// Mitsubishi GX Works2 project: 5   PLC: FX3U/FX3UC

// task Task_01 (event TRUE, interval 0, priority 31): POU_01

PROGRAM POU_01
VAR
  cnt : INT;
  wstep : INT;
  ton1 : TON;
END_VAR
Y0 := M0 XOR M1 XOR M2;
END_PROGRAM
